# EPICS alarm handler configuration: epics_alh/alarms_list_StatusMonitor.alhConfig
GROUP NULL StatusMonitor
